FUNCTION_BLOCK PUBLIC Load3Station
VAR_INPUT
END_VAR
VAR_OUTPUT
END_VAR
VAR
	xTrigger :BOOL := FALSE; // triggers processing
	State : eLoadSta3State := eLoadSta3State.eUnknown;
	NextState : eLoadSta3State := eLoadSta3State.eUnknown;
	bFirst : BOOL := TRUE;
	VUT : BYTE; //VehicleID Under Station
	DwellTimer : TON;
	LoadingComplete : BOOL := FALSE;
	CycleNumb: INT := 0;
	RowNumber :INT:=0;
	SeedNumber : INT:=5;
END_VAR

IF (GVL_IO.MachineEStopped) THEN 
	State := eLoadSta3State.eUnknown;
	NextState := eLoadSta3State.eUnknown;
END_IF

CASE State OF
eLoadSta3State.eUnknown:
	NextState := eLoadSta3State.eReady;

eLoadSta3State.eInit:

eLoadSta3State.eHoming:

eLoadSta3State.eReady:

IF (xTrigger) THEN
		NextState := eLoadSta3State.eWaitForLoadComplete;
		
		DwellTimer(IN:=FALSE);	
	END_IF

eLoadSta3State.eDwell:

eLoadSta3State.eWaitForLoadComplete:
	 IF (LoadingComplete) THEN
		NextState := eLoadSta3State.eDepart;
		UpdatePartData();
		LoadingComplete := FALSE;
		DwellTimer(IN:=FALSE);
	END_IF


eLoadSta3State.eProcessing:

eLoadSta3State.eDepart:
	Stations.fbRoutePlanner.M_NotifyVehStaCmpl(StationIndex:= MM_CONST.LOAD_3_STA, VehicleID := VUT);
	xTrigger := FALSE;
    IF (Stations.fbCycleControl.StopRequested) THEN
		NextState := eLoadSta3State.eStopActive;
	ELSE	
		NextState := eLoadSta3State.eReady;	
	END_IF

eLoadSta3State.eStopActive:
	IF (NOT Stations.fbCycleControl.StopRequested) THEN
		NextState := eLoadSta3State.eReady;
	END_IF
	
eLoadSta3State.eError:

END_CASE

IF (State <> NextState) THEN
	bFirst := TRUE;
ELSE
	bFirst := FALSE;
END_IF

State := NextState;
Status.StationsState[MM_CONST.LOAD_3_STA_HMI_STATE] := State;

METHOD PUBLIC ClearVehicleTrigger : BOOL
VAR_INPUT
END_VAR
xTrigger := FALSE;
END_METHOD

PROPERTY PUBLIC LoadComplete : BOOL
SET
LoadingComplete := LoadComplete;
END_SET
END_PROPERTY

METHOD PUBLIC ResetState : BOOL
VAR_INPUT
END_VAR
	State := eLoadSta3State.eUnknown;
	NextState := eLoadSta3State.eUnknown;
END_METHOD

METHOD PUBLIC SetRowNumber : BOOL
VAR_INPUT
	RowLocationNumber : INT;
END_VAR
RowNumber := RowLocationNumber;
END_METHOD

PROPERTY PUBLIC Trigger : BOOL
SET
xTrigger := Trigger;
END_SET
END_PROPERTY

METHOD PUBLIC UpdatePartData : BOOL
VAR_INPUT
END_VAR
memset(ADR(PartsData.Status[VUT]),0,SIZEOF(PartDataType));
PartsData.Status[VUT].LoadTime := SYSTEMTIME_TO_STRING(Logging.fbCurrTime.systemTime);
//PartsData.Status[VUT].CavityNumber := 9 + (CycleNumb MOD 4);
PartsData.Status[VUT].CavityNumber := RowNumber + SeedNumber;
CycleNumb := CycleNumb+1; // Use this till Yushin Robot sends out this information with Bit Location ID
PartsData.Status[VUT].OverallStatus := ePartStatus.eLoaded; // At least that is the assumption. We may want to check on how to turn off cavities later, but this will be caught by vision.
PartsData.Status[VUT].BarrelSize := LotsData.Lot.BarrelSize; // we are copying this data in case we might in future want to have more than one lots running at the same time on the machine
PartsData.Status[VUT].PartNumber := LotsData.Lot.PartNumber; // we are copying this data in case we might in future want to have more than one lots running at the same time on the machine
PartsData.Status[VUT].LotNumber := LotsData.Lot.LotNumber; // we are copying this data in case we might in future want to have more than one lots running at the same time on the machine
END_METHOD

PROPERTY PUBLIC VehicleUnderTest : BYTE
GET
VehicleUnderTest := VUT;
END_GET
SET
VUT := VehicleUnderTest;
END_SET
END_PROPERTY

END_FUNCTION_BLOCK

(* stored: Version 1.1.0.1, ProductVersion 3.1.4022.3
   POU Load3Station: Id {4a5e7ad5-a119-43a8-bc76-42db68c9d77f}, SpecialFunc None
   Method ClearVehicleTrigger: Id {481820c8-5859-40c1-9315-3ddae5c64382}
   Property LoadComplete: Id {4b308fe3-127b-4bed-88a4-377988e22c6d}
   Set Set: Id {3954f32e-8f2e-43f7-a525-c4d5163288c9}
   Method ResetState: Id {e931cf68-a211-48b1-9fe1-9d8fc26f62ef}
   Method SetRowNumber: Id {eb7a373d-2701-42dd-a51b-669104ecc2cb}
   Property Trigger: Id {79a6d11b-9300-449f-81ad-dcfbb183056d}
   Set Set: Id {48e7e57f-2e67-49a2-a7ce-40c0816f4ee4}
   Method UpdatePartData: Id {83b8a77f-498f-4bef-bf21-10807c4c852d}
   Property VehicleUnderTest: Id {3dd97944-f448-4c5a-b17d-b61059f40103}
   Get Get: Id {23050b32-c4b9-41c2-8d54-770554ef09bf}
   Set Set: Id {046fffc1-eee1-45b2-bb63-35bab2a08368} *)
